// TIA Portal V20 export
TYPE "LWONIK_typeZoneStatus"
// stored: Access Published
   STRUCT
      safetyReleased1 : Bool;
      safetyReleased2 : Bool;
      ackReq : Bool;
      safetyFault : Bool;
      highSpeedEnable : Bool;
      activeSLS : Bool;
      activeSTO : Bool;
      activeSOS : Bool;
      activeSS1 : Bool;
      activeSS2 : Bool;
      allFDoorClose : Bool;
      sFDoorOpen : Bool;
      mFDoorOpen : Bool;
      STKCVCoverNOK1 : Bool;   // STK1 Safety Conveyor Cover Status
      STKCVCoverNOK2 : Bool;   // STK2 Safety Conveyor Cover Status
      STKCVCoverAllOK : Bool;   // All STK Safety Conveyor Cover Status
   END_STRUCT;
END_TYPE
